// TwinCAT 3 PLC project PLC_1
// ProgramVersion: 3.1.4024.0
// libraries:
//   Tc2_Standard, * (Beckhoff Automation GmbH)
//   Tc2_System, * (Beckhoff Automation GmbH)
//   Tc3_Module, * (Beckhoff Automation GmbH)
// project tree:
//   GVLs/ GVL.TcGVL
//   / PlcTask.TcTTO
//   POUs/ ButtonController.TcPOU, MAIN.TcPOU
// real-time tasks:
//   TASK PlcTask: cycle T#10ms, priority 20, ADS port 350
//   TASK PlcTask1: cycle T#10ms, priority 21, ADS port 351

CONFIGURATION PLC_1
    RESOURCE PLC ON TwinCAT3
        TASK PlcTask(INTERVAL := T#10ms, PRIORITY := 21);
        PROGRAM MAIN WITH PlcTask : MAIN;
    END_RESOURCE
END_CONFIGURATION

// ---- GVLs/GVL.TcGVL
{attribute 'qualified_only'}
VAR_GLOBAL
	mb_Input_Coils : ARRAY [0..3] OF BOOL;
	mb_Output_Coils : ARRAY [0..7] OF BOOL;
END_VAR

// ---- POUs/MAIN.TcPOU
PROGRAM MAIN
VAR
	ButtonController : ButtonController;
END_VAR

ButtonController();

END_PROGRAM

// ---- POUs/ButtonController.TcPOU
FUNCTION_BLOCK ButtonController
VAR_INPUT
	Start : BOOL;
	Reset : BOOL;
	Stop : BOOL;
	EmergencyStop : BOOL;
END_VAR
VAR_OUTPUT
	StartLight : BOOL;
	ResetLight : BOOL;
	StopLight : BOOL;
END_VAR
VAR
	tBlink : TON;
	BlinkBit : BOOL;
	state : INT;
END_VAR

// I/O assignment
GVL.mb_Input_Coils[1] := StartLight;
GVL.mb_Input_Coils[2] := ResetLight;
GVL.mb_Input_Coils[3] := StopLight;
Start := gvl.mb_Output_Coils[3];
Reset := gvl.mb_Output_Coils[4];
Stop := gvl.mb_Output_Coils[5];
EmergencyStop := gvl.mb_Output_Coils[7];
//
// Blinking logic
tBlink(IN := NOT tBlink.Q, PT := T#1000MS);
BlinkBit := tBlink.ET > T#500MS;
//
CASE state OF
	0: // Idle (stop)
		StartLight := BlinkBit;
		StopLight := TRUE;
		ResetLight := FALSE;
		IF Start THEN
			state := 1;
		END_IF;
		IF NOT EmergencyStop THEN
			state := 2;
		END_IF;
	1: // Running state
		StartLight := TRUE;
		StopLight := FALSE;
		ResetLight := FALSE;
		IF NOT EmergencyStop THEN
			state := 2;
		END_IF;
		IF NOT Stop THEN
			state := 0;
		END_IF;
	2: // Emergency Stop
		StopLight := TRUE;
		StartLight := FALSE;
		IF EmergencyStop THEN
			ResetLight := BlinkBit;
			IF Reset THEN
				state := 3;
			END_IF;
		ELSE
			ResetLight := FALSE;
		END_IF;
	3: // After emergency stop
		StopLight := FALSE;
		ResetLight := TRUE;
		StartLight := BlinkBit;
		IF Start THEN
			state := 1;
		END_IF;
		IF NOT EmergencyStop THEN
			state := 2;
		END_IF;
ELSE
	state := 0;
END_CASE;

END_FUNCTION_BLOCK
